Fanuc KAREL source: ks00033.KL

-- PROVISIONAL review KL for V940-1; original PC SHA256 4091559107272818415468b2126f8a44374841240a2de58c02ae9fd49a816e53
-- Incomplete behavior may be omitted. Consult companion uncertainty JSON. Do not deploy.
PROGRAM KS00033
%NOLOCKGROUP
VAR
  FLAG : BOOLEAN
  N : INTEGER
  STATUS : INTEGER
  PN : STRING[80]
  VN : STRING[80]
-- UNRESOLVED_DECL A type=00201c
-- UNRESOLVED_DECL B type=00201c
BEGIN
  -- V9_ZERO_TABLE_METADATA_HINT layout=0001; no indexed target words; source/name/runtime held
  -- UNRESOLVED_PC offsets 5-13; opcodes 3F,75
  -- UNRESOLVED_PC offsets 18-27; opcodes 3F,75
  -- UNRESOLVED_PC offsets 32-45; opcodes 22,1D,23
  -- UNRESOLVED_PC offsets 50-54; opcodes 7F
END KS00033
